Yaskawa INFORM job: TEST4.JBI

/JOB
//NAME TEST4
///FOLDERNAME INNE
//POS
///NPOS 55,55,55,2,0,0
///TOOL 0
///POSTYPE PULSE
///PULSE
C00000=172153,-78771,-99140,22114,121919,-58523
C00001=172147,-80104,-70575,18948,104742,-61737
C00002=174896,-83252,-68987,19218,101642,-61221
C00003=176341,-84638,-68086,19378,100101,-60941
C00004=175260,-82760,-67286,19221,100804,-61223
C00005=176341,-85165,-69579,19426,100714,-60841
C00006=184166,-72684,-62736,20865,100859,-57926
C00007=182742,-71414,-63608,20759,102335,-58194
C00008=180008,-68528,-65144,20588,105303,-58692
C00009=180015,-63882,-92048,24291,122904,-55038
C00010=-208366,-104906,-99424,-22310,104158,50067
C00011=-208386,-99487,-80688,-21594,96012,51577
C00012=-212429,-100514,-78057,-21964,92940,50658
C00013=-214096,-100759,-76935,-22118,91734,50271
C00014=-221445,-103969,-78075,-22785,88854,48132
C00015=-221451,-102416,-74939,-22785,87805,48330
C00016=-221445,-103969,-78075,-22785,88854,48132
C00017=-214096,-100759,-76935,-22118,91734,50271
C00018=-208643,-117028,-77166,-25577,77313,51874
C00019=-213005,-118978,-77715,-25773,75395,50674
C00020=-208643,-117028,-77166,-25577,77313,51874
C00021=-208822,-120108,-82491,-25446,78796,51482
C00022=-206641,-120588,-83865,-25326,79996,52031
C00023=-201308,-121362,-87158,-24990,83076,53347
C00024=-201283,-134020,-108014,-24879,88851,52142
C00025=-205406,-141653,-121151,-23339,95635,50994
C00026=-205450,-120231,-85125,-23161,85322,52980
C00027=-210644,-119757,-81866,-23654,82247,51698
C00028=-213321,-119294,-80159,-23891,80745,51026
C00029=-213318,-120376,-81809,-23866,81167,50942
C00030=-211152,-118332,-79886,-23715,81657,51632
C00031=-218171,-102372,-74847,-23930,84339,48526
C00032=-215903,-102696,-76483,-23811,85763,49074
C00033=-211453,-102932,-79591,-23563,88685,50129
C00034=-211417,-111920,-112059,-24427,102801,47286
C00035=198520,-284271,-144991,39803,12344,-29978
C00036=198453,-180882,-95123,14695,32927,-18090
C00037=204349,-170581,-90734,11023,34679,-14762
C00038=206608,-165588,-88484,9639,35596,-13505
C00039=204068,-167604,-88597,11099,34923,-14866
C00040=206612,-167644,-90281,9626,35644,-13497
C00041=194152,-162294,-88248,14700,38740,-19065
C00042=191199,-167071,-90535,16215,38215,-20585
C00043=183866,-176858,-95019,19834,37429,-24323
C00044=183904,-275380,-144574,38041,19440,-33430
C00045=119359,-302859,-143845,-57887,26972,62937
C00046=119482,-192117,-94856,-32072,46909,48828
C00047=119556,-185650,-90671,-31707,47570,48609
C00048=119590,-182551,-88579,-31561,47842,48522
C00049=119576,-184941,-90377,-31619,47733,48556
C00050=131934,-182427,-88590,-30575,51399,52075
C00051=119957,-176935,-88821,-30217,50570,47709
C00052=119940,-179932,-90933,-30316,50356,47775
C00053=119903,-186185,-95162,-30573,49816,47944
C00054=119821,-294547,-145016,-50255,30103,59220
BC00000=398174,15,1075175
BC00001=398174,15,1075175
BC00002=398174,15,1075175
BC00003=398174,15,1075175
BC00004=398174,15,1075175
BC00005=398174,15,1075175
BC00006=398174,15,1075175
BC00007=398174,15,1075175
BC00008=398174,15,1075175
BC00009=398174,15,1075175
BC00010=398174,15,1075175
BC00011=398174,15,1075175
BC00012=398174,15,1075175
BC00013=398174,15,1075175
BC00014=398174,15,1075175
BC00015=398174,15,1075175
BC00016=398174,15,1075175
BC00017=398174,15,1075175
BC00018=398174,15,1075175
BC00019=398174,15,1075175
BC00020=398174,15,1075175
BC00021=398174,15,1075175
BC00022=398174,15,1075175
BC00023=398174,15,1075175
BC00024=398174,15,1075175
BC00025=398174,15,1075175
BC00026=398174,15,1075175
BC00027=398174,15,1075175
BC00028=398174,15,1075175
BC00029=398174,15,1075175
BC00030=398174,15,1075175
BC00031=398174,15,1075175
BC00032=398174,15,1075175
BC00033=398174,15,1075175
BC00034=398174,15,1075175
BC00035=398174,15,1075175
BC00036=398174,15,1075175
BC00037=398174,15,1075175
BC00038=398174,15,1075175
BC00039=398174,15,1075175
BC00040=398174,15,1075175
BC00041=398174,15,1075175
BC00042=398174,15,1075175
BC00043=398174,15,1075175
BC00044=398174,15,1075175
BC00045=238383,15,1075175
BC00046=238383,15,1075175
BC00047=243989,15,1075175
BC00048=246792,15,1075175
BC00049=246792,15,1075175
BC00050=246792,15,1075175
BC00051=246792,15,1075175
BC00052=243989,15,1075175
BC00053=238383,15,1075175
BC00054=238383,15,1075175
EC00000=-1596313,1112951
EC00001=-1596313,1112951
EC00002=-1596313,1112951
EC00003=-1596313,1112951
EC00004=-1596313,1112951
EC00005=-1596313,1112951
EC00006=-1596313,1112951
EC00007=-1596313,1112951
EC00008=-1596313,1112951
EC00009=-1596313,1112951
EC00010=-1596313,1112951
EC00011=-1596313,1112951
EC00012=-1596313,1112951
EC00013=-1596313,1112951
EC00014=-1596313,1112951
EC00015=-1596313,1112951
EC00016=-1596313,1112951
EC00017=-1596313,1112951
EC00018=-1596313,1112951
EC00019=-1596313,1112951
EC00020=-1596313,1112951
EC00021=-1596313,1112951
EC00022=-1596313,1112951
EC00023=-1596313,1112951
EC00024=-1596313,1112951
EC00025=-1596313,1112951
EC00026=-1596313,1112951
EC00027=-1596313,1112951
EC00028=-1596313,1112951
EC00029=-1596313,1112951
EC00030=-1596313,1112951
EC00031=-1596313,1112951
EC00032=-1596313,1112951
EC00033=-1596313,1112951
EC00034=-1596313,1112951
EC00035=-1596313,1112951
EC00036=-1596313,1112951
EC00037=-1596313,1112951
EC00038=-1596313,1112951
EC00039=-1596313,1112951
EC00040=-1596313,1112951
EC00041=-1596313,1112951
EC00042=-1596313,1112951
EC00043=-1596313,1112951
EC00044=-1596313,1112951
EC00045=-1596313,1112951
EC00046=-1596313,1112951
EC00047=-1596313,1112951
EC00048=-1596313,1112951
EC00049=-1596313,1112951
EC00050=-1596313,1112951
EC00051=-1596313,1112951
EC00052=-1596313,1112951
EC00053=-1596313,1112951
EC00054=-1596313,1112951
///POSTYPE BASE
///RECTAN
///RCONF 0,0,0,0,1,0,0,0,0,0,0,0,0,0,0,0,0,0,0,0,0,0,0,0
P00006=2.006,1.622,-0.565,0.0000,0.0000,0.0000
P00021=0.073,2.058,-0.109,0.0000,0.0000,0.0000
//INST
///DATE 2023/10/04 15:16
///ATTR SC,RW
///GROUP1 RB1,BS1
///GROUP2 ST1
NOP
'test4
'Path W777
SSFTOF
MOVJ C00000 BC00000 VJ=100.00  +MOVJ EC00000 VJ=100.00
SSFTON P021
SMOVL C00001 BC00001 V=1000.0  +MOVJ EC00001
SMOVL C00002 BC00002 V=400.0  +MOVJ EC00002
SMOVL C00003 BC00003 V=100.0 PL=0  +MOVJ EC00003
SREFP 1 C00004 BC00004  +REFP EC00004
SREFP 2 C00005 BC00005  +REFP EC00005
ARCON ASF#(4)
WVON WEV#(4)
SMOVL C00006 BC00006 V=10.0  +MOVJ EC00006
ARCOF AEF#(1)
WVOF
SMOVL C00007 BC00007 V=400.0  +MOVJ EC00007
SMOVL C00008 BC00008 V=1000.0  +MOVJ EC00008
SMOVL C00009 BC00009 V=1000.0  +MOVJ EC00009
SSFTOF
'Path S781 (for W778)
SSFTOF
MOVJ C00010 BC00010 VJ=100.00  +MOVJ EC00010 VJ=100.00
MOVL C00011 BC00011 V=1000.0  +MOVJ EC00011 VJ=100.00
MOVL C00012 BC00012 V=400.0  +MOVJ EC00012 VJ=100.00
SMOVL C00013 BC00013 V=100.0  +MOVJ EC00013
SMOVL C00014 BC00014 V=60.0  +MOVJ EC00014
SREFP 3 C00015 BC00015  +REFP EC00015
CALL JOB:SEARCH-R1-S1
SET P021 P006
SSFTON P021
SMOVL C00016 BC00016 V=60.0  +MOVJ EC00016
SMOVL C00017 BC00017 V=100.0  +MOVJ EC00017
SMOVL C00018 BC00018 V=60.0  +MOVJ EC00018
SREFP 3 C00019 BC00019  +REFP EC00019
CALL JOB:SEARCH-R1-S1
SET P021 P006
SSFTON P021
SMOVL C00020 BC00020 V=60.0  +MOVJ EC00020
SMOVL C00021 BC00021 V=100.0  +MOVJ EC00021
MOVL C00022 BC00022 V=400.0  +MOVJ EC00022 VJ=100.00
MOVL C00023 BC00023 V=1000.0  +MOVJ EC00023 VJ=100.00
MOVL C00024 BC00024 V=1000.0  +MOVJ EC00024 VJ=100.00
'Path W778
SSFTOF
MOVJ C00025 BC00025 VJ=100.00  +MOVJ EC00025 VJ=100.00
SSFTON P021
SMOVL C00026 BC00026 V=1000.0  +MOVJ EC00026
SMOVL C00027 BC00027 V=400.0  +MOVJ EC00027
SMOVL C00028 BC00028 V=100.0 PL=0  +MOVJ EC00028
SREFP 1 C00029 BC00029  +REFP EC00029
SREFP 2 C00030 BC00030  +REFP EC00030
ARCON ASF#(4)
WVON WEV#(4)
SMOVL C00031 BC00031 V=10.0  +MOVJ EC00031
ARCOF AEF#(1)
WVOF
SMOVL C00032 BC00032 V=400.0  +MOVJ EC00032
SMOVL C00033 BC00033 V=1000.0  +MOVJ EC00033
SMOVL C00034 BC00034 V=1000.0  +MOVJ EC00034
SSFTOF
'Path W779
SSFTOF
MOVJ C00035 BC00035 VJ=100.00  +MOVJ EC00035 VJ=100.00
MOVL C00036 BC00036 V=1000.0  +MOVJ EC00036 VJ=100.00
MOVL C00037 BC00037 V=400.0  +MOVJ EC00037 VJ=100.00
SMOVL C00038 BC00038 V=100.0 PL=0  +MOVJ EC00038
SREFP 1 C00039 BC00039  +REFP EC00039
SREFP 2 C00040 BC00040  +REFP EC00040
ARCON ASF#(4)
WVON WEV#(4)
SMOVL C00041 BC00041 V=10.0  +MOVJ EC00041
ARCOF AEF#(1)
WVOF
MOVL C00042 BC00042 V=400.0  +MOVJ EC00042 VJ=100.00
MOVL C00043 BC00043 V=1000.0  +MOVJ EC00043 VJ=100.00
MOVL C00044 BC00044 V=1000.0  +MOVJ EC00044 VJ=100.00
'Path W780
SSFTOF
MOVJ C00045 BC00045 VJ=100.00  +MOVJ EC00045 VJ=100.00
MOVL C00046 BC00046 V=1000.0  +MOVJ EC00046 VJ=100.00
MOVL C00047 BC00047 V=400.0  +MOVJ EC00047 VJ=100.00
SMOVL C00048 BC00048 V=100.0 PL=0  +MOVJ EC00048
SREFP 1 C00049 BC00049  +REFP EC00049
SREFP 2 C00050 BC00050  +REFP EC00050
ARCON ASF#(4)
WVON WEV#(4)
SMOVL C00051 BC00051 V=10.0  +MOVJ EC00051
ARCOF AEF#(1)
WVOF
MOVL C00052 BC00052 V=400.0  +MOVJ EC00052 VJ=100.00
MOVL C00053 BC00053 V=1000.0  +MOVJ EC00053 VJ=100.00
MOVL C00054 BC00054 V=1000.0  +MOVJ EC00054 VJ=100.00
END
